{attribute 'qualified_only'}
{attribute 'strict'}
{attribute 'to_string'}
TYPE eGensetMode :
(
	Isochronous := 0,
	Droop := 1,
	FixedPower := 2
);
END_TYPE

(* stored: Version 1.1.0.1, ProductVersion 3.1.4026.18
   DUT eGensetMode: Id {07709d88-d6c2-4c81-9bb0-3162e7f3fc71} *)
